LIN {X 0,Y 43.603,Z 528.429,A -85,B 0,C 180,E1 -29830.157,E2 -29830.157} C_VEL
LIN {X 0,Y 50.48,Z 525.546,A -85,B 0,C 180,E1 -29839.984,E2 -29839.984} C_VEL
LIN {X 0,Y 58.397,Z 521.621,A -85,B 0,C 180,E1 -29847.411,E2 -29847.411} C_VEL
LIN {X 0,Y 65.879,Z 517.271,A -85,B 0,C 180,E1 -29852.356,E2 -29852.356} C_VEL
LIN {X 0,Y 66.634,Z 516.529,A -85,B 0,C 180,E1 -29853.877,E2 -29853.877} C_VEL
LIN {X 0,Y 50.194,Z 523.456,A -85,B 0,C 180,E1 -29891.406,E2 -29891.406} C_VEL
LIN {X 0,Y 53.552,Z 526.244,A -85,B 0,C 180,E1 -29913.828,E2 -29913.828} C_VEL
LIN {X 0,Y 52.648,Z 527.165,A -85,B 0,C 180,E1 -29916.768,E2 -29916.768} C_VEL
LIN {X 0,Y 47.505,Z 529.474,A -85,B 0,C 180,E1 -29922.28,E2 -29922.28} C_VEL
LIN {X 0,Y 42.937,Z 531.358,A -85,B 0,C 180,E1 -29929.089,E2 -29929.089} C_VEL
LIN {X 0,Y 39.15,Z 532.78,A -85,B 0,C 180,E1 -29937.403,E2 -29937.403} C_VEL
LIN {X 0,Y 34.788,Z 534.418,A -85,B 0,C 180,E1 -29958.333,E2 -29958.333} C_VEL
LIN {X 0,Y 34.425,Z 534.642,A -85,B 0,C 180,E1 -29969.988,E2 -29969.988} C_VEL
LIN {X 0,Y 34.526,Z 534.386,A -85,B 0,C 180,E1 -29981.733,E2 -29981.733} C_VEL
LIN {X 0,Y 38.456,Z 532.695,A -85,B 0,C 180,E1 -30003.235,E2 -30003.235} C_VEL
LIN {X 0,Y 42.036,Z 531.228,A -85,B 0,C 180,E1 -30011.958,E2 -30011.958} C_VEL
LIN {X 0,Y 48.96,Z 528.221,A -85,B 0,C 180,E1 -30022.125,E2 -30022.125} C_VEL
LIN {X 0,Y 56.997,Z 524.156,A -85,B 0,C 180,E1 -30029.656,E2 -30029.656} C_VEL
LIN {X 0,Y 67.244,Z 517.902,A -85,B 0,C 180,E1 -30036.119,E2 -30036.119} C_VEL
LIN {X 0,Y 76.549,Z 511.099,A -85,B 0,C 180,E1 -30040.214,E2 -30040.214} C_VEL
LIN {X 0,Y 86.203,Z 502.606,A -85,B 0,C 180,E1 -30043.311,E2 -30043.311} C_VEL
LIN {X 0,Y 94.436,Z 493.887,A -85,B 0,C 180,E1 -30045.328,E2 -30045.328} C_VEL
LIN {X 0,Y 102.768,Z 483.16,A -85,B 0,C 180,E1 -30047.019,E2 -30047.019} C_VEL
LIN {X 0,Y 109.493,Z 472.34,A -85,B 0,C 180,E1 -30048.174,E2 -30048.174} C_VEL
LIN {X 0,Y 115.534,Z 460.022,A -85,B 0,C 180,E1 -30049.058,E2 -30049.058} C_VEL
LIN {X 0,Y 120.064,Z 447.665,A -85,B 0,C 180,E1 -30049.674,E2 -30049.674} C_VEL
LIN {X 0,Y 123.277,Z 434.898,A -85,B 0,C 180,E1 -30050.113,E2 -30050.113} C_VEL
LIN {X 0,Y 123.771,Z 432.175,A -85,B 0,C 180,E1 -30050.295,E2 -30050.295} C_VEL
LIN {X 0,Y 123.051,Z 429.181,A -85,B 0,C 180,E1 -30054.264,E2 -30054.264} C_VEL
LIN {X 0,Y 122.801,Z 426.596,A -85,B 0,C 180,E1 -30059.18,E2 -30059.18} C_VEL
LIN {X 0,Y 122.776,Z 426.735,A -85,B 0,C 180,E1 -30061.435,E2 -30061.435} C_VEL
LIN {X 0,Y 123.208,Z 430.114,A -85,B 0,C 180,E1 -30067.626,E2 -30067.626} C_VEL
LIN {X 0,Y 123.67,Z 432.48,A -85,B 0,C 180,E1 -30070.503,E2 -30070.503} C_VEL
LIN {X 0,Y 120.488,Z 445.463,A -85,B 0,C 180,E1 -30071.113,E2 -30071.113} C_VEL
LIN {X 0,Y 116.334,Z 457.129,A -85,B 0,C 180,E1 -30071.832,E2 -30071.832} C_VEL
LIN {X 0,Y 110.872,Z 468.748,A -85,B 0,C 180,E1 -30072.961,E2 -30072.961} C_VEL
LIN {X 0,Y 104.234,Z 479.778,A -85,B 0,C 180,E1 -30074.267,E2 -30074.267} C_VEL
LIN {X 0,Y 96.853,Z 489.734,A -85,B 0,C 180,E1 -30075.974,E2 -30075.974} C_VEL
LIN {X 0,Y 95.525,Z 491.286,A -85,B 0,C 180,E1 -30076.298,E2 -30076.298} C_VEL
LIN {X 0,Y 91.566,Z 495.586,A -85,B 0,C 180,E1 -30076.913,E2 -30076.913} C_VEL
LIN {X 0,Y 84.241,Z 502.258,A -85,B 0,C 180,E1 -30077.082,E2 -30077.082} C_VEL
LIN {X 0,Y 76.426,Z 508.335,A -85,B 0,C 180,E1 -30077.395,E2 -30077.395} C_VEL
LIN {X 0,Y 71.727,Z 511.663,A -85,B 0,C 180,E1 -30078.425,E2 -30078.425} C_VEL
LIN {X 0,Y 61.017,Z 518.479,A -85,B 0,C 180,E1 -30082.879,E2 -30082.879} C_VEL
LIN {X 0,Y 51.981,Z 523.199,A -85,B 0,C 180,E1 -30088.516,E2 -30088.516} C_VEL
LIN {X 0,Y 43.55,Z 526.802,A -85,B 0,C 180,E1 -30096.223,E2 -30096.223} C_VEL
LIN {X 0,Y 38.489,Z 528.654,A -85,B 0,C 180,E1 -30103.096,E2 -30103.096} C_VEL
LIN {X 0,Y 34.088,Z 530.059,A -85,B 0,C 180,E1 -30111.807,E2 -30111.807} C_VEL
LIN {X 0,Y 28.409,Z 531.645,A -85,B 0,C 180,E1 -30135.692,E2 -30135.692} C_VEL
LIN {X 0,Y 27.647,Z 531.869,A -85,B 0,C 180,E1 -30150.015,E2 -30150.015} C_VEL
LIN {X 0,Y 28.408,Z 531.669,A -85,B 0,C 180,E1 -30164.338,E2 -30164.338} C_VEL
LIN {X 0,Y 34.047,Z 530.118,A -85,B 0,C 180,E1 -30188.277,E2 -30188.277} C_VEL
LIN {X 0,Y 38.462,Z 528.745,A -85,B 0,C 180,E1 -30196.977,E2 -30196.977} C_VEL
LIN {X 0,Y 46.246,Z 525.861,A -85,B 0,C 180,E1 -30206.719,E2 -30206.719} C_VEL
LIN {X 0,Y 54.895,Z 521.936,A -85,B 0,C 180,E1 -30213.676,E2 -30213.676} C_VEL
LIN {X 0,Y 56.082,Z 521.07,A -85,B 0,C 180,E1 -30216.108,E2 -30216.108} C_VEL
LIN {X 0,Y 43.6,Z 526.705,A -85,B 0,C 180,E1 -30258.807,E2 -30258.807} C_VEL
LIN {X 0,Y 44.849,Z 527.607,A -85,B 0,C 180,E1 -30268.041,E2 -30268.041} C_VEL
LIN {X 0,Y 44.818,Z 528.488,A -85,B 0,C 180,E1 -30273.517,E2 -30273.517} C_VEL
LIN {X 0,Y 37.858,Z 531.042,A -85,B 0,C 180,E1 -30282.035,E2 -30282.035} C_VEL
LIN {X 0,Y 33.382,Z 532.463,A -85,B 0,C 180,E1 -30290.817,E2 -30290.817} C_VEL
LIN {X 0,Y 27.878,Z 534.102,A -85,B 0,C 180,E1 -30315.384,E2 -30315.384} C_VEL
LIN {X 0,Y 27.331,Z 534.325,A -85,B 0,C 180,E1 -30329.985,E2 -30329.985} C_VEL
LIN {X 0,Y 27.6,Z 534.068,A -85,B 0,C 180,E1 -30344.737,E2 -30344.737} C_VEL
LIN {X 0,Y 32.705,Z 532.375,A -85,B 0,C 180,E1 -30370.124,E2 -30370.124} C_VEL
LIN {X 0,Y 37.04,Z 530.909,A -85,B 0,C 180,E1 -30379.356,E2 -30379.356} C_VEL
LIN {X 0,Y 44.923,Z 527.901,A -85,B 0,C 180,E1 -30389.348,E2 -30389.348} C_VEL
LIN {X 0,Y 53.731,Z 523.835,A -85,B 0,C 180,E1 -30396.272,E2 -30396.272} C_VEL
LIN {X 0,Y 64.678,Z 517.583,A -85,B 0,C 180,E1 -30401.928,E2 -30401.928} C_VEL
LIN {X 0,Y 74.435,Z 510.781,A -85,B 0,C 180,E1 -30405.395,E2 -30405.395} C_VEL
LIN {X 0,Y 84.434,Z 502.29,A -85,B 0,C 180,E1 -30407.942,E2 -30407.942} C_VEL
LIN {X 0,Y 92.891,Z 493.573,A -85,B 0,C 180,E1 -30409.571,E2 -30409.571} C_VEL
LIN {X 0,Y 100.554,Z 484.009,A -85,B 0,C 180,E1 -30410.809,E2 -30410.809} C_VEL
LIN {X 0,Y 107.401,Z 473.557,A -85,B 0,C 180,E1 -30411.754,E2 -30411.754} C_VEL
LIN {X 0,Y 113.426,Z 461.906,A -85,B 0,C 180,E1 -30412.441,E2 -30412.441} C_VEL
LIN {X 0,Y 118.293,Z 449.516,A -85,B 0,C 180,E1 -30412.962,E2 -30412.962} C_VEL
LIN {X 0,Y 121.758,Z 437.047,A -85,B 0,C 180,E1 -30413.371,E2 -30413.371} C_VEL
LIN {X 0,Y 121.558,Z 435.773,A -85,B 0,C 180,E1 -30415.44,E2 -30415.44} C_VEL
LIN {X 0,Y 121.574,Z 433.463,A -85,B 0,C 180,E1 -30420,E2 -30420} C_VEL
LIN {X 0,Y 121.41,Z 434.971,A -85,B 0,C 180,E1 -30423.319,E2 -30423.319} C_VEL
LIN {X 0,Y 121.585,Z 436.863,A -85,B 0,C 180,E1 -30426.851,E2 -30426.851} C_VEL
LIN {X 0,Y 121.616,Z 437.202,A -85,B 0,C 180,E1 -30427.335,E2 -30427.335} C_VEL
LIN {X 0,Y 118.01,Z 449.753,A -85,B 0,C 180,E1 -30427.986,E2 -30427.986} C_VEL
LIN {X 0,Y 113.73,Z 460.539,A -85,B 0,C 180,E1 -30428.636,E2 -30428.636} C_VEL
LIN {X 0,Y 107.798,Z 472.108,A -85,B 0,C 180,E1 -30429.593,E2 -30429.593} C_VEL
LIN {X 0,Y 100.178,Z 483.627,A -85,B 0,C 180,E1 -30430.858,E2 -30430.858} C_VEL
LIN {X 0,Y 91.804,Z 493.859,A -85,B 0,C 180,E1 -30432.581,E2 -30432.581} C_VEL
LIN {X 0,Y 82.243,Z 503.271,A -85,B 0,C 180,E1 -30435.06,E2 -30435.06} C_VEL
LIN {X 0,Y 72.156,Z 511.367,A -85,B 0,C 180,E1 -30438.279,E2 -30438.279} C_VEL
LIN {X 0,Y 71.727,Z 511.663,A -85,B 0,C 180,E1 -30438.425,E2 -30438.425} C_VEL
LIN {X 0,Y 66.896,Z 514.82,A -85,B 0,C 180,E1 -30439.614,E2 -30439.614} C_VEL
LIN {X 0,Y 54.63,Z 521.173,A -85,B 0,C 180,E1 -30440.853,E2 -30440.853} C_VEL
LIN {X 0,Y 47.499,Z 524.215,A -85,B 0,C 180,E1 -30442.519,E2 -30442.519} C_VEL
LIN {X 0,Y 44.123,Z 525.525,A -85,B 0,C 180,E1 -30444.381,E2 -30444.381} C_VEL
LIN {X 0,Y 34.045,Z 528.971,A -85,B 0,C 180,E1 -30454.359,E2 -30454.359} C_VEL
LIN {X 0,Y 28.848,Z 530.376,A -85,B 0,C 180,E1 -30463.063,E2 -30463.063} C_VEL
LIN {X 0,Y 21.614,Z 531.962,A -85,B 0,C 180,E1 -30491.045,E2 -30491.045} C_VEL
LIN {X 0,Y 20.555,Z 532.186,A -85,B 0,C 180,E1 -30510.02,E2 -30510.02} C_VEL
LIN {X 0,Y 21.614,Z 531.985,A -85,B 0,C 180,E1 -30528.995,E2 -30528.995} C_VEL
LIN {X 0,Y 28.823,Z 530.434,A -85,B 0,C 180,E1 -30557.033,E2 -30557.033} C_VEL
LIN {X 0,Y 34.011,Z 529.061,A -85,B 0,C 180,E1 -30565.767,E2 -30565.767} C_VEL
LIN {X 0,Y 42.763,Z 526.177,A -85,B 0,C 180,E1 -30574.698,E2 -30574.698} C_VEL
LIN {X 0,Y 45.849,Z 524.966,A -85,B 0,C 180,E1 -30576.905,E2 -30576.905} C_VEL
LIN {X 0,Y 44.273,Z 525.208,A -85,B 0,C 180,E1 -30581.489,E2 -30581.489} C_VEL
LIN {X 0,Y 37.054,Z 528.936,A -85,B 0,C 180,E1 -30622.292,E2 -30622.292} C_VEL
LIN {X 0,Y 37.404,Z 529.174,A -85,B 0,C 180,E1 -30625.406,E2 -30625.406} C_VEL
LIN {X 0,Y 37.112,Z 529.612,A -85,B 0,C 180,E1 -30628.888,E2 -30628.888} C_VEL
LIN {X 0,Y 28.238,Z 532.147,A -85,B 0,C 180,E1 -30641.678,E2 -30641.678} C_VEL
LIN {X 0,Y 21.079,Z 533.785,A -85,B 0,C 180,E1 -30670.504,E2 -30670.504} C_VEL
LIN {X 0,Y 20.221,Z 534.007,A -85,B 0,C 180,E1 -30689.98,E2 -30689.98} C_VEL
LIN {X 0,Y 20.784,Z 533.75,A -85,B 0,C 180,E1 -30709.743,E2 -30709.743} C_VEL
LIN {X 0,Y 27.623,Z 532.055,A -85,B 0,C 180,E1 -30739.731,E2 -30739.731} C_VEL
LIN {X 0,Y 32.846,Z 530.59,A -85,B 0,C 180,E1 -30748.832,E2 -30748.832} C_VEL
LIN {X 0,Y 41.734,Z 527.581,A -85,B 0,C 180,E1 -30757.822,E2 -30757.822} C_VEL
LIN {X 0,Y 51.272,Z 523.516,A -85,B 0,C 180,E1 -30763.61,E2 -30763.61} C_VEL
LIN {X 0,Y 62.834,Z 517.265,A -85,B 0,C 180,E1 -30768.118,E2 -30768.118} C_VEL
LIN {X 0,Y 72.965,Z 510.464,A -85,B 0,C 180,E1 -30770.815,E2 -30770.815} C_VEL
LIN {X 0,Y 83.236,Z 501.974,A -85,B 0,C 180,E1 -30772.753,E2 -30772.753} C_VEL
LIN {X 0,Y 91.872,Z 493.259,A -85,B 0,C 180,E1 -30773.928,E2 -30773.928} C_VEL
LIN {X 0,Y 99.668,Z 483.698,A -85,B 0,C 180,E1 -30774.834,E2 -30774.834} C_VEL
LIN {X 0,Y 106.614,Z 473.249,A -85,B 0,C 180,E1 -30775.538,E2 -30775.538} C_VEL
LIN {X 0,Y 112.713,Z 461.603,A -85,B 0,C 180,E1 -30776.013,E2 -30776.013} C_VEL
LIN {X 0,Y 117.725,Z 448.96,A -85,B 0,C 180,E1 -30776.406,E2 -30776.406} C_VEL
LIN {X 0,Y 119.771,Z 442.247,A -85,B 0,C 180,E1 -30776.636,E2 -30776.636} C_VEL
LIN {X 0,Y 119.931,Z 440.535,A -85,B 0,C 180,E1 -30780,E2 -30780} C_VEL
LIN {X 0,Y 119.646,Z 442.423,A -85,B 0,C 180,E1 -30784.177,E2 -30784.177} C_VEL
LIN {X 0,Y 115.956,Z 453.552,A -85,B 0,C 180,E1 -30784.704,E2 -30784.704} C_VEL
LIN {X 0,Y 111.162,Z 464.444,A -85,B 0,C 180,E1 -30785.318,E2 -30785.318} C_VEL
LIN {X 0,Y 104.255,Z 476.588,A -85,B 0,C 180,E1 -30786.147,E2 -30786.147} C_VEL
LIN {X 0,Y 96.517,Z 487.245,A -85,B 0,C 180,E1 -30787.235,E2 -30787.235} C_VEL
LIN {X 0,Y 88.82,Z 495.927,A -85,B 0,C 180,E1 -30788.51,E2 -30788.51} C_VEL
LIN {X 0,Y 80.173,Z 504.031,A -85,B 0,C 180,E1 -30790.304,E2 -30790.304} C_VEL
LIN {X 0,Y 70.257,Z 511.683,A -85,B 0,C 180,E1 -30792.782,E2 -30792.782} C_VEL
LIN {X 0,Y 61.929,Z 516.954,A -85,B 0,C 180,E1 -30795.313,E2 -30795.313} C_VEL
LIN {X 0,Y 52.149,Z 522.095,A -85,B 0,C 180,E1 -30799.399,E2 -30799.399} C_VEL
LIN {X 0,Y 44.123,Z 525.525,A -85,B 0,C 180,E1 -30804.381,E2 -30804.381} C_VEL
LIN {X 0,Y 38.983,Z 527.337,A -85,B 0,C 180,E1 -30807.545,E2 -30807.545} C_VEL
LIN {X 0,Y 29.768,Z 529.749,A -85,B 0,C 180,E1 -30812.208,E2 -30812.208} C_VEL
LIN {X 0,Y 22.431,Z 531.188,A -85,B 0,C 180,E1 -30818.394,E2 -30818.394} C_VEL
LIN {X 0,Y 17.02,Z 532.03,A -85,B 0,C 180,E1 -30830.831,E2 -30830.831} C_VEL
LIN {X 0,Y 16.436,Z 532.044,A -85,B 0,C 180,E1 -30833.546,E2 -30833.546} C_VEL
LIN {X 0,Y 13.482,Z 532.502,A -85,B 0,C 180,E1 -30870.03,E2 -30870.03} C_VEL
LIN {X 0,Y 15.081,Z 532.302,A -85,B 0,C 180,E1 -30897.806,E2 -30897.806} C_VEL
LIN {X 0,Y 24.538,Z 530.751,A -85,B 0,C 180,E1 -30929.262,E2 -30929.262} C_VEL
LIN {X 0,Y 34.337,Z 528.347,A -85,B 0,C 180,E1 -30940.071,E2 -30940.071} C_VEL
LIN {X 0,Y 35.591,Z 527.932,A -85,B 0,C 180,E1 -30942.643,E2 -30942.643} C_VEL
LIN {X 0,Y 29.919,Z 530.368,A -85,B 0,C 180,E1 -30979.977,E2 -30979.977} C_VEL
LIN {X 0,Y 24.111,Z 531.831,A -85,B 0,C 180,E1 -30988.987,E2 -30988.987} C_VEL
LIN {X 0,Y 14.57,Z 533.467,A -85,B 0,C 180,E1 -31021.129,E2 -31021.129} C_VEL
LIN {X 0,Y 13.109,Z 533.69,A -85,B 0,C 180,E1 -31049.969,E2 -31049.969} C_VEL
LIN {X 0,Y 14.268,Z 533.43,A -85,B 0,C 180,E1 -31079.476,E2 -31079.476} C_VEL
LIN {X 0,Y 23.639,Z 531.735,A -85,B 0,C 180,E1 -31113.075,E2 -31113.075} C_VEL
LIN {X 0,Y 29.79,Z 530.272,A -85,B 0,C 180,E1 -31120.635,E2 -31120.635} C_VEL
LIN {X 0,Y 39.595,Z 527.262,A -85,B 0,C 180,E1 -31127.436,E2 -31127.436} C_VEL
LIN {X 0,Y 51.908,Z 522.165,A -85,B 0,C 180,E1 -31132.219,E2 -31132.219} C_VEL
LIN {X 0,Y 63.488,Z 515.937,A -85,B 0,C 180,E1 -31134.978,E2 -31134.978} C_VEL
LIN {X 0,Y 73.914,Z 508.854,A -85,B 0,C 180,E1 -31136.633,E2 -31136.633} C_VEL
LIN {X 0,Y 84.389,Z 500.048,A -85,B 0,C 180,E1 -31137.825,E2 -31137.825} C_VEL
LIN {X 0,Y 93.145,Z 491.017,A -85,B 0,C 180,E1 -31138.495,E2 -31138.495} C_VEL
LIN {X 0,Y 101.034,Z 480.977,A -85,B 0,C 180,E1 -31139.029,E2 -31139.029} C_VEL
LIN {X 0,Y 108.053,Z 469.869,A -85,B 0,C 180,E1 -31139.451,E2 -31139.451} C_VEL
LIN {X 0,Y 113.952,Z 457.969,A -85,B 0,C 180,E1 -31139.706,E2 -31139.706} C_VEL
LIN {X 0,Y 117.508,Z 448.625,A -85,B 0,C 180,E1 -31139.861,E2 -31139.861} C_VEL
LIN {X 0,Y 117.873,Z 447.564,A -85,B 0,C 180,E1 -31140,E2 -31140} C_VEL
LIN {X 0,Y 117.77,Z 447.829,A -85,B 0,C 180,E1 -31140.855,E2 -31140.855} C_VEL
LIN {X 0,Y 116.495,Z 451.464,A -85,B 0,C 180,E1 -31141.131,E2 -31141.131} C_VEL
LIN {X 0,Y 111.603,Z 463.034,A -85,B 0,C 180,E1 -31141.557,E2 -31141.557} C_VEL
LIN {X 0,Y 105.484,Z 474.118,A -85,B 0,C 180,E1 -31142.115,E2 -31142.115} C_VEL
LIN {X 0,Y 97.626,Z 485.395,A -85,B 0,C 180,E1 -31142.839,E2 -31142.839} C_VEL
LIN {X 0,Y 89.789,Z 494.486,A -85,B 0,C 180,E1 -31143.72,E2 -31143.72} C_VEL
LIN {X 0,Y 80.971,Z 502.869,A -85,B 0,C 180,E1 -31144.98,E2 -31144.98} C_VEL
LIN {X 0,Y 70.755,Z 510.793,A -85,B 0,C 180,E1 -31146.698,E2 -31146.698} C_VEL
LIN {X 0,Y 60.446,Z 517.271,A -85,B 0,C 180,E1 -31148.823,E2 -31148.823} C_VEL
LIN {X 0,Y 50.238,Z 522.413,A -85,B 0,C 180,E1 -31151.73,E2 -31151.73} C_VEL
LIN {X 0,Y 40.251,Z 526.374,A -85,B 0,C 180,E1 -31156.23,E2 -31156.23} C_VEL
LIN {X 0,Y 30.601,Z 529.289,A -85,B 0,C 180,E1 -31163.305,E2 -31163.305} C_VEL
LIN {X 0,Y 24.564,Z 530.693,A -85,B 0,C 180,E1 -31170.902,E2 -31170.902} C_VEL
LIN {X 0,Y 16.436,Z 532.044,A -85,B 0,C 180,E1 -31193.546,E2 -31193.546} C_VEL
LIN {X 0,Y 13.305,Z 532.462,A -85,B 0,C 180,E1 -31212.931,E2 -31212.931} C_VEL
LIN {X 0,Y 11.273,Z 532.603,A -85,B 0,C 180,E1 -31239.289,E2 -31239.289} C_VEL
LIN {X 0,Y 14.849,Z 532.094,A -85,B 0,C 180,E1 -31291.77,E2 -31291.77} C_VEL
LIN {X 0,Y 19.695,Z 531.41,A -85,B 0,C 180,E1 -31303.284,E2 -31303.284} C_VEL
LIN {X 0,Y 21.533,Z 531.103,A -85,B 0,C 180,E1 -31305.297,E2 -31305.297} C_VEL
LIN {X 0,Y 23.4,Z 530.783,A -85,B 0,C 180,E1 -31306.863,E2 -31306.863} C_VEL
LIN {X 0,Y 25.195,Z 530.415,A -85,B 0,C 180,E1 -31310.815,E2 -31310.815} C_VEL
LIN {X 0,Y 23.71,Z 530.831,A -85,B 0,C 180,E1 -31319.999,E2 -31319.999} C_VEL
LIN {X 0,Y 21.552,Z 531.507,A -85,B 0,C 180,E1 -31331.871,E2 -31331.871} C_VEL
LIN {X 0,Y 14.971,Z 532.526,A -85,B 0,C 180,E1 -31340.062,E2 -31340.062} C_VEL
LIN {X 0,Y 9.03,Z 533.15,A -85,B 0,C 180,E1 -31358.827,E2 -31358.827} C_VEL
LIN {X 0,Y 5.982,Z 533.371,A -85,B 0,C 180,E1 -31409.933,E2 -31409.933} C_VEL
LIN {X 0,Y 8.794,Z 533.112,A -85,B 0,C 180,E1 -31462.977,E2 -31462.977} C_VEL
LIN {X 0,Y 21.375,Z 531.416,A -85,B 0,C 180,E1 -31490.418,E2 -31490.418} C_VEL
LIN {X 0,Y 28.24,Z 529.954,A -85,B 0,C 180,E1 -31494.394,E2 -31494.394} C_VEL
LIN {X 0,Y 38.675,Z 526.943,A -85,B 0,C 180,E1 -31497.807,E2 -31497.807} C_VEL
LIN {X 0,Y 50.573,Z 522.241,A -85,B 0,C 180,E1 -31500,E2 -31500} C_VEL
LIN {X 0,Y 63.264,Z 515.619,A -85,B 0,C 180,E1 -31501.432,E2 -31501.432} C_VEL
LIN {X 0,Y 63.271,Z 515.607,A -85,B 0,C 180,E1 -31501.667,E2 -31501.667} C_VEL
LIN {X 0,Y 52.429,Z 521.306,A -85,B 0,C 180,E1 -31503.124,E2 -31503.124} C_VEL
LIN {X 0,Y 42.336,Z 525.478,A -85,B 0,C 180,E1 -31505.222,E2 -31505.222} C_VEL
LIN {X 0,Y 35.415,Z 527.754,A -85,B 0,C 180,E1 -31507.236,E2 -31507.236} C_VEL
LIN {X 0,Y 28.547,Z 529.606,A -85,B 0,C 180,E1 -31510.102,E2 -31510.102} C_VEL
LIN {X 0,Y 21.786,Z 531.01,A -85,B 0,C 180,E1 -31514.658,E2 -31514.658} C_VEL
LIN {X 0,Y 9.411,Z 532.595,A -85,B 0,C 180,E1 -31541.751,E2 -31541.751} C_VEL
LIN {X 0,Y 6.398,Z 532.818,A -85,B 0,C 180,E1 -31590.063,E2 -31590.063} C_VEL
LIN {X 0,Y 9.417,Z 532.618,A -85,B 0,C 180,E1 -31638.339,E2 -31638.339} C_VEL
LIN {X 0,Y 21.533,Z 531.103,A -85,B 0,C 180,E1 -31665.297,E2 -31665.297} C_VEL
LIN {X 0,Y 23.702,Z 533.084,A -85,B 0,C 180,E1 -31667.011,E2 -31667.011} C_VEL
LIN {X 0,Y 23.702,Z 600,A -85,B 0,C 180,E1 -31667.011,E2 -31667.011} C_VEL
LIN {X 0,Y 23.702,Z 600,A -85,B 0,C 180,E1 -31667.011,E2 -31667.011}

QRS_NEXT_CUT()

QRS_NEXT()
QRS_HOME()

END
